{attribute 'GeneratedUsingTerminal: EL2535-0103-0023'}
{attribute addProperty BoxType "EL2535-0103-0023"}
{attribute addProperty Id "EtcSlaveTerminalBasePWM_Status_Channel_1AT %I*PWM_Status_Channel_77939B114PWM_Status_Channel_2AT %I*PWM_Status_Channel_77939B114PWM_Control_Channel_1AT %Q*PWM_Control_Channel_63F162E45PWM_Control_Channel_2AT %Q*PWM_Control_Channel_63F162E45WcStateAT %I*WcState_9091E0EB2InfoDataAT %I*InfoData_32EB74EA10"}
{attribute addProperty CRC "3466088981"}
{attribute addProperty Size "30"}
TYPE EL2535_CE985215 EXTENDS EtcSlaveTerminalBase :
STRUCT
	{attribute addProperty Name "PWM_Status_Channel_1"}
	PWM_Status_Channel_1 : PWM_Status_Channel_77939B11;
	{attribute addProperty Name "PWM_Status_Channel_2"}
	PWM_Status_Channel_2 : PWM_Status_Channel_77939B11;
	{attribute addProperty Name "PWM_Control_Channel_1"}
	PWM_Control_Channel_1 : PWM_Control_Channel_63F162E4;
	{attribute addProperty Name "PWM_Control_Channel_2"}
	PWM_Control_Channel_2 : PWM_Control_Channel_63F162E4;
	{attribute addProperty Name "WcState"}
	WcState : WcState_9091E0EB;
	{attribute addProperty Name "InfoData"}
	InfoData : InfoData_32EB74EA;
END_STRUCT
END_TYPE

(* stored: Version 1.2.0.0, ProductVersion 3.1.4024.9
   DUT EL2535_CE985215: Id {aeacee0c-3c2c-4272-afaf-bb7e42c65eb4} *)
